(* Logix 5000 project; controller Generic 1768-L43 rev 15.6; software revision 15.01; part 4 of 10 *)
(* tags used below, declared in another part *)
   EL_CTRL_7 : UDT_AxisHistory_CTRL;
   EL_CTRL_8 : UDT_AxisHistory_CTRL;
   EventLog_N7 : UDT_AxisHistory_DLM[51];
   EventLog_N8 : UDT_AxisHistory_DLM[51];
   LogLength : DINT;
   Motion_Group : ALIAS FOR MotionGroup;
   Servo_Axis_Node_7 : ALIAS FOR AXIS_Servo_Generic;
   Servo_Axis_Node_8 : ALIAS FOR AXIS_Servo_Generic;
(* AXIS_EventLog, continued *)

ROUTINE R07_EventLog_Node7   (* ladder *)
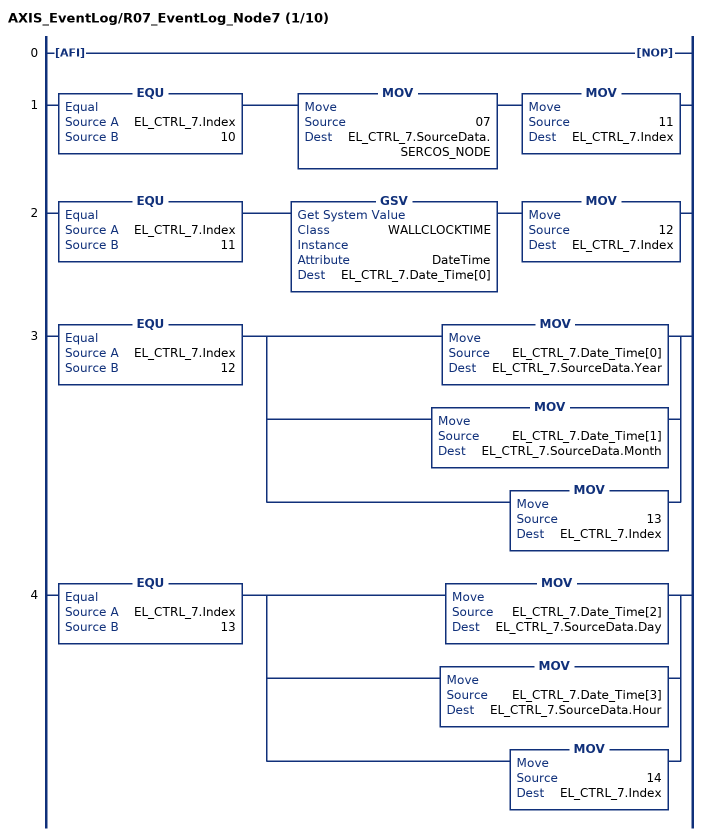
   0: AFI()NOP();
   1: EQU(EL_CTRL_7.Index,10)MOV(07,EL_CTRL_7.SourceData.SERCOS_NODE)MOV(11,EL_CTRL_7.Index);
   2: EQU(EL_CTRL_7.Index,11)GSV(WALLCLOCKTIME,,DateTime,EL_CTRL_7.Date_Time[0])MOV(12,EL_CTRL_7.Index);
   3: EQU(EL_CTRL_7.Index,12)[MOV(EL_CTRL_7.Date_Time[0],EL_CTRL_7.SourceData.Year) ,MOV(EL_CTRL_7.Date_Time[1],EL_CTRL_7.SourceData.Month) ,MOV(13,EL_CTRL_7.Index) ];
   4: EQU(EL_CTRL_7.Index,13)[MOV(EL_CTRL_7.Date_Time[2],EL_CTRL_7.SourceData.Day) ,MOV(EL_CTRL_7.Date_Time[3],EL_CTRL_7.SourceData.Hour) ,MOV(14,EL_CTRL_7.Index) ];
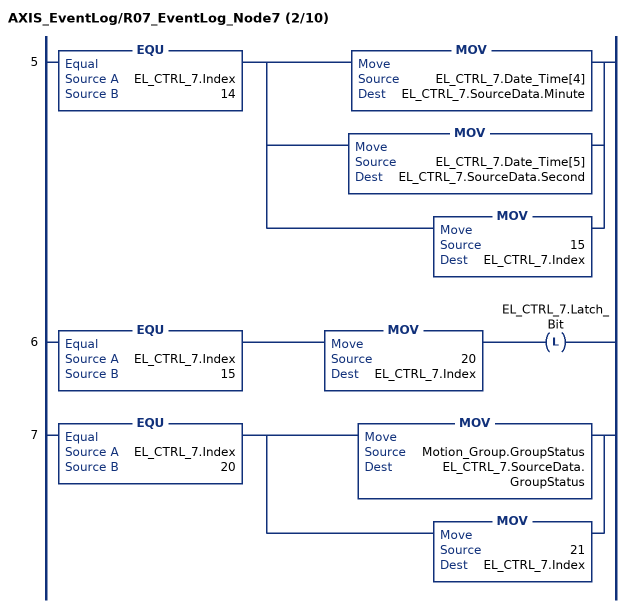
   5: EQU(EL_CTRL_7.Index,14)[MOV(EL_CTRL_7.Date_Time[4],EL_CTRL_7.SourceData.Minute) ,MOV(EL_CTRL_7.Date_Time[5],EL_CTRL_7.SourceData.Second) ,MOV(15,EL_CTRL_7.Index) ];
   6: EQU(EL_CTRL_7.Index,15)MOV(20,EL_CTRL_7.Index)OTL(EL_CTRL_7.Latch_Bit);
   7: EQU(EL_CTRL_7.Index,20)[MOV(Motion_Group.GroupStatus,EL_CTRL_7.SourceData.GroupStatus) ,MOV(21,EL_CTRL_7.Index) ];
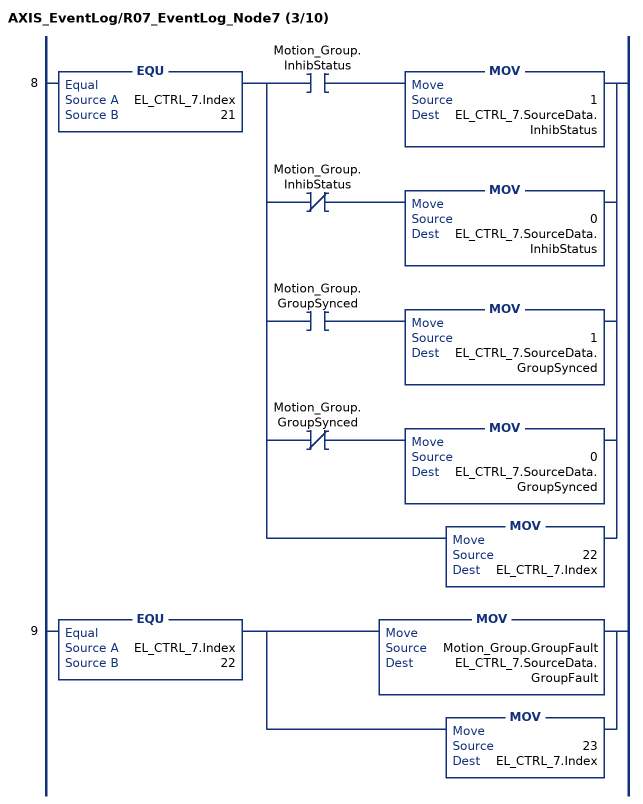
   8: EQU(EL_CTRL_7.Index,21)[XIC(Motion_Group.InhibStatus) MOV(1,EL_CTRL_7.SourceData.InhibStatus) ,XIO(Motion_Group.InhibStatus) MOV(0,EL_CTRL_7.SourceData.InhibStatus) ,XIC(Motion_Group.GroupSynced) MOV(1,EL_CTRL_7.SourceData.GroupSynced) ,XIO(Motion_Group.GroupSynced) MOV(0,EL_CTRL_7.SourceData.GroupSynced) ,MOV(22,EL_CTRL_7.Index) ];
   9: EQU(EL_CTRL_7.Index,22)[MOV(Motion_Group.GroupFault,EL_CTRL_7.SourceData.GroupFault) ,MOV(23,EL_CTRL_7.Index) ];
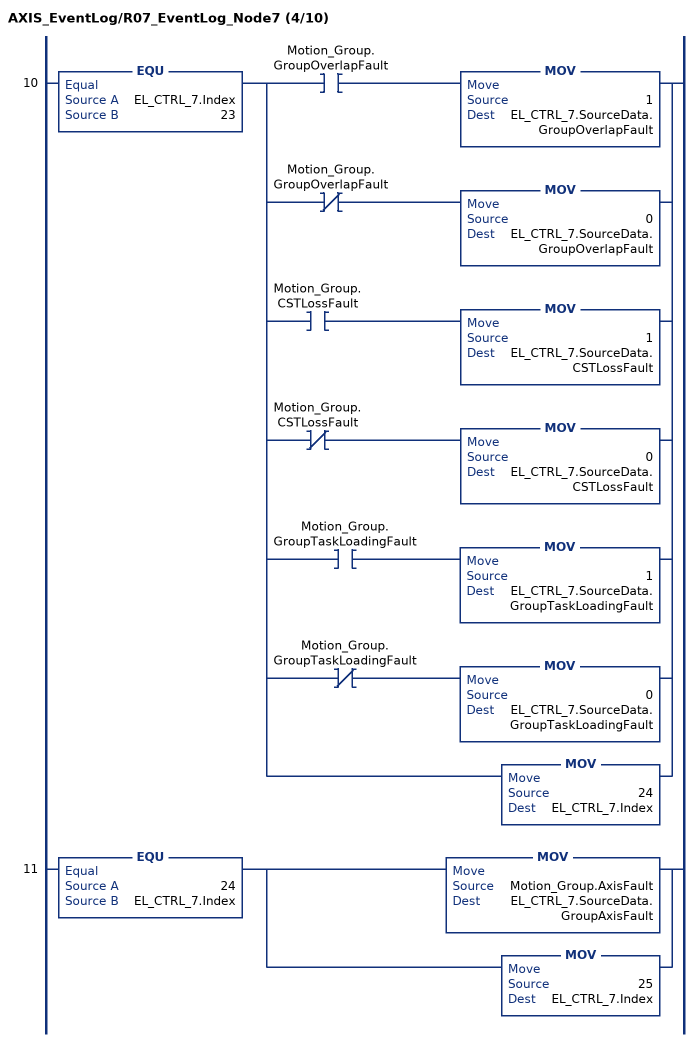
   10: EQU(EL_CTRL_7.Index,23)[XIC(Motion_Group.GroupOverlapFault) MOV(1,EL_CTRL_7.SourceData.GroupOverlapFault) ,XIO(Motion_Group.GroupOverlapFault) MOV(0,EL_CTRL_7.SourceData.GroupOverlapFault) ,XIC(Motion_Group.CSTLossFault) MOV(1,EL_CTRL_7.SourceData.CSTLossFault) ,XIO(Motion_Group.CSTLossFault) MOV(0,EL_CTRL_7.SourceData.CSTLossFault) ,XIC(Motion_Group.GroupTaskLoadingFault) MOV(1,EL_CTRL_7.SourceData.GroupTaskLoadingFault) ,XIO(Motion_Group.GroupTaskLoadingFault) MOV(0,EL_CTRL_7.SourceData.GroupTaskLoadingFault) ,MOV(24,EL_CTRL_7.Index) ];
   11: EQU(24,EL_CTRL_7.Index)[MOV(Motion_Group.AxisFault,EL_CTRL_7.SourceData.GroupAxisFault) ,MOV(25,EL_CTRL_7.Index) ];
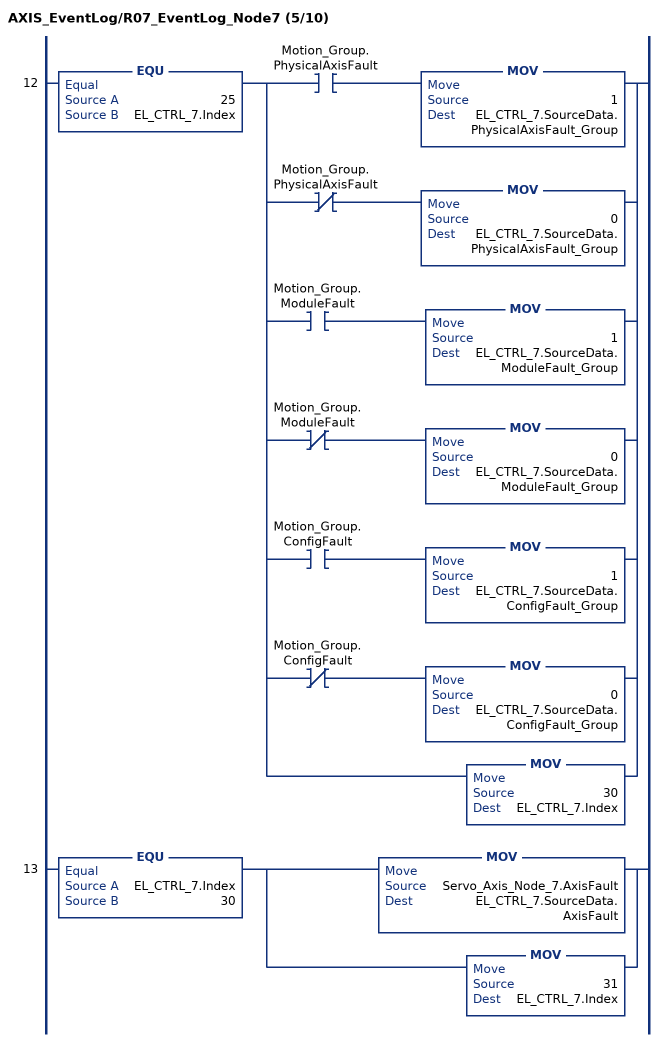
   12: EQU(25,EL_CTRL_7.Index)[XIC(Motion_Group.PhysicalAxisFault) MOV(1,EL_CTRL_7.SourceData.PhysicalAxisFault_Group) ,XIO(Motion_Group.PhysicalAxisFault) MOV(0,EL_CTRL_7.SourceData.PhysicalAxisFault_Group) ,XIC(Motion_Group.ModuleFault) MOV(1,EL_CTRL_7.SourceData.ModuleFault_Group) ,XIO(Motion_Group.ModuleFault) MOV(0,EL_CTRL_7.SourceData.ModuleFault_Group) ,XIC(Motion_Group.ConfigFault) MOV(1,EL_CTRL_7.SourceData.ConfigFault_Group) ,XIO(Motion_Group.ConfigFault) MOV(0,EL_CTRL_7.SourceData.ConfigFault_Group) ,MOV(30,EL_CTRL_7.Index) ];
   13: EQU(EL_CTRL_7.Index,30)[MOV(Servo_Axis_Node_7.AxisFault,EL_CTRL_7.SourceData.AxisFault) ,MOV(31,EL_CTRL_7.Index) ];
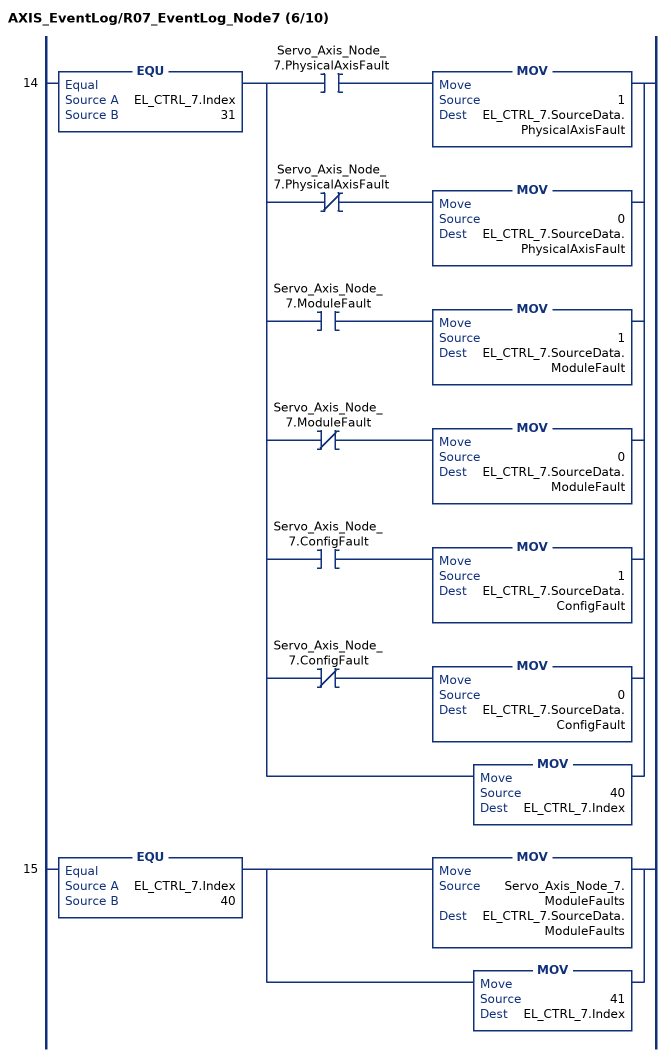
   14: EQU(EL_CTRL_7.Index,31)[XIC(Servo_Axis_Node_7.PhysicalAxisFault) MOV(1,EL_CTRL_7.SourceData.PhysicalAxisFault) ,XIO(Servo_Axis_Node_7.PhysicalAxisFault) MOV(0,EL_CTRL_7.SourceData.PhysicalAxisFault) ,XIC(Servo_Axis_Node_7.ModuleFault) MOV(1,EL_CTRL_7.SourceData.ModuleFault) ,XIO(Servo_Axis_Node_7.ModuleFault) MOV(0,EL_CTRL_7.SourceData.ModuleFault) ,XIC(Servo_Axis_Node_7.ConfigFault) MOV(1,EL_CTRL_7.SourceData.ConfigFault) ,XIO(Servo_Axis_Node_7.ConfigFault) MOV(0,EL_CTRL_7.SourceData.ConfigFault) ,MOV(40,EL_CTRL_7.Index) ];
   15: EQU(EL_CTRL_7.Index,40)[MOV(Servo_Axis_Node_7.ModuleFaults,EL_CTRL_7.SourceData.ModuleFaults) ,MOV(41,EL_CTRL_7.Index) ];
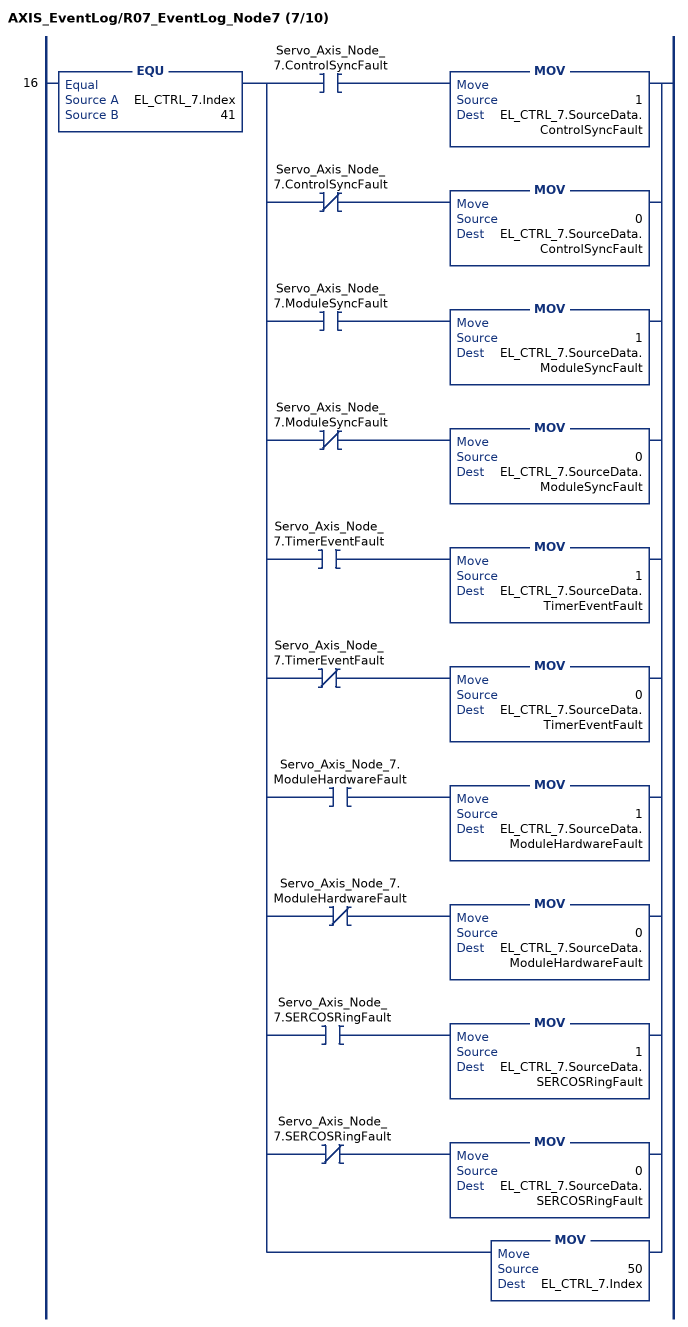
   16: EQU(EL_CTRL_7.Index,41)[XIC(Servo_Axis_Node_7.ControlSyncFault) MOV(1,EL_CTRL_7.SourceData.ControlSyncFault) ,XIO(Servo_Axis_Node_7.ControlSyncFault) MOV(0,EL_CTRL_7.SourceData.ControlSyncFault) ,XIC(Servo_Axis_Node_7.ModuleSyncFault) MOV(1,EL_CTRL_7.SourceData.ModuleSyncFault) ,XIO(Servo_Axis_Node_7.ModuleSyncFault) MOV(0,EL_CTRL_7.SourceData.ModuleSyncFault) ,XIC(Servo_Axis_Node_7.TimerEventFault) MOV(1,EL_CTRL_7.SourceData.TimerEventFault) ,XIO(Servo_Axis_Node_7.TimerEventFault) MOV(0,EL_CTRL_7.SourceData.TimerEventFault) ,XIC(Servo_Axis_Node_7.ModuleHardwareFault) MOV(1,EL_CTRL_7.SourceData.ModuleHardwareFault) ,XIO(Servo_Axis_Node_7.ModuleHardwareFault) MOV(0,EL_CTRL_7.SourceData.ModuleHardwareFault) ,XIC(Servo_Axis_Node_7.SERCOSRingFault) MOV(1,EL_CTRL_7.SourceData.SERCOSRingFault) ,XIO(Servo_Axis_Node_7.SERCOSRingFault) MOV(0,EL_CTRL_7.SourceData.SERCOSRingFault) ,MOV(50,EL_CTRL_7.Index) ];
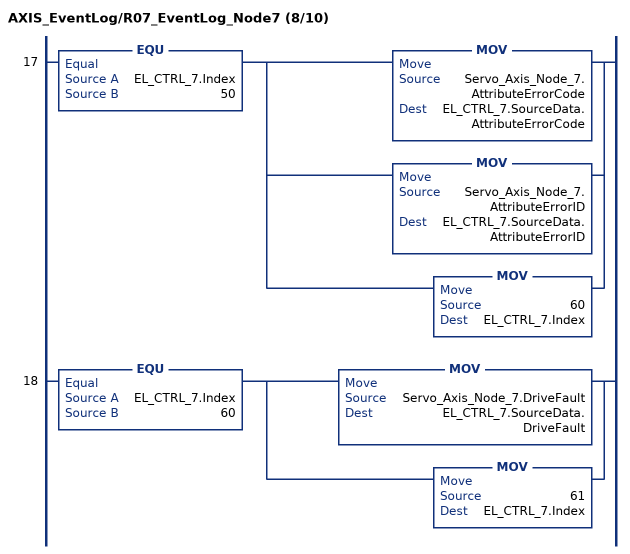
   17: EQU(EL_CTRL_7.Index,50)[MOV(Servo_Axis_Node_7.AttributeErrorCode,EL_CTRL_7.SourceData.AttributeErrorCode) ,MOV(Servo_Axis_Node_7.AttributeErrorID,EL_CTRL_7.SourceData.AttributeErrorID) ,MOV(60,EL_CTRL_7.Index) ];
   18: EQU(EL_CTRL_7.Index,60)[MOV(Servo_Axis_Node_7.DriveFault,EL_CTRL_7.SourceData.DriveFault) ,MOV(61,EL_CTRL_7.Index) ];
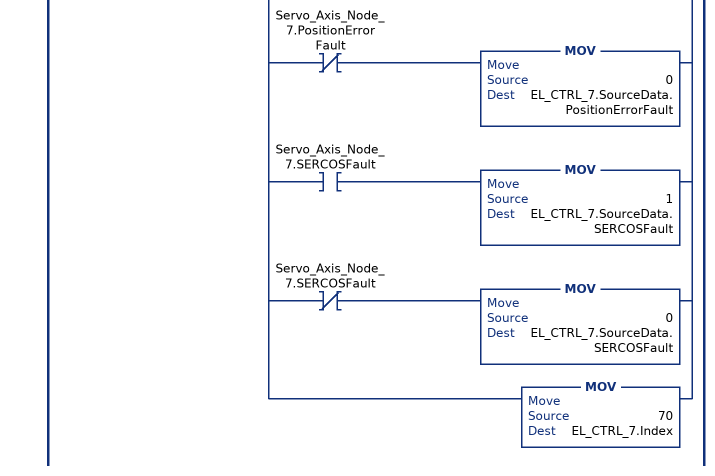
   19: EQU(EL_CTRL_7.Index,61)[XIC(Servo_Axis_Node_7.PosSoftOvertravelFault) MOV(1,EL_CTRL_7.SourceData.PosSoftOvertravelFault) ,XIO(Servo_Axis_Node_7.PosSoftOvertravelFault) MOV(0,EL_CTRL_7.SourceData.PosSoftOvertravelFault) ,XIC(Servo_Axis_Node_7.NegSoftOvertravelFault) MOV(1,EL_CTRL_7.SourceData.NegSoftOvertravelFault) ,XIO(Servo_Axis_Node_7.NegSoftOvertravelFault) MOV(0,EL_CTRL_7.SourceData.NegSoftOvertravelFault) ,XIC(Servo_Axis_Node_7.PosHardOvertravelFault) MOV(1,EL_CTRL_7.SourceData.PosHardOvertravelFault) ,XIO(Servo_Axis_Node_7.PosHardOvertravelFault) MOV(0,EL_CTRL_7.SourceData.PosHardOvertravelFault) ,XIC(Servo_Axis_Node_7.NegHardOvertravelFault) MOV(1,EL_CTRL_7.SourceData.NegHardOvertravelFault) ,XIO(Servo_Axis_Node_7.NegHardOvertravelFault) MOV(0,EL_CTRL_7.SourceData.NegHardOvertravelFault) ,XIC(Servo_Axis_Node_7.MotFeedbackFault) MOV(1,EL_CTRL_7.SourceData.MotFeedbackFault) ,XIO(Servo_Axis_Node_7.MotFeedbackFault) MOV(0,EL_CTRL_7.SourceData.MotFeedbackFault) ,XIC(Servo_Axis_Node_7.MotFeedbackNoiseFault) MOV(1,EL_CTRL_7.SourceData.MotFeedbackNoiseFault) ,XIO(Servo_Axis_Node_7.MotFeedbackNoiseFault) MOV(0,EL_CTRL_7.SourceData.MotFeedbackNoiseFault) ,XIC(Servo_Axis_Node_7.AuxFeedbackFault) MOV(1,EL_CTRL_7.SourceData.AuxFeedbackFault) ,XIO(Servo_Axis_Node_7.AuxFeedbackFault) MOV(0,EL_CTRL_7.SourceData.AuxFeedbackFault) ,XIC(Servo_Axis_Node_7.AuxFeedbackNoiseFault) MOV(1,EL_CTRL_7.SourceData.AuxFeedbackNoiseFault) ,XIO(Servo_Axis_Node_7.AuxFeedbackNoiseFault) MOV(0,EL_CTRL_7.SourceData.AuxFeedbackNoiseFault) ,XIC(Servo_Axis_Node_7.DriveEnableInputFault) MOV(1,EL_CTRL_7.SourceData.DriveEnableInputFault) ,XIO(Servo_Axis_Node_7.DriveEnableInputFault) MOV(0,EL_CTRL_7.SourceData.DriveEnableInputFault) ,XIC(Servo_Axis_Node_7.CommonBusFault) MOV(1,EL_CTRL_7.SourceData.CommonBusFault) ,XIO(Servo_Axis_Node_7.CommonBusFault) MOV(0,EL_CTRL_7.SourceData.CommonBusFault) ,XIC(Servo_Axis_Node_7.PreChargeOverloadFault) MOV(1,EL_CTRL_7.SourceData.PreChargeOverloadFault) ,XIO(Servo_Axis_Node_7.PreChargeOverloadFault) MOV(0,EL_CTRL_7.SourceData.PreChargeOverloadFault) ,XIC(Servo_Axis_Node_7.GroundShortFault) MOV(1,EL_CTRL_7.SourceData.GroundShortFault) ,XIO(Servo_Axis_Node_7.GroundShortFault) MOV(0,EL_CTRL_7.SourceData.GroundShortFault) ,XIC(Servo_Axis_Node_7.DriveHardFault) MOV(1,EL_CTRL_7.SourceData.DriveHardFault) ,XIO(Servo_Axis_Node_7.DriveHardFault) MOV(0,EL_CTRL_7.SourceData.DriveHardFault) ,XIC(Servo_Axis_Node_7.OverSpeedFault) MOV(1,EL_CTRL_7.SourceData.OverSpeedFault) ,XIO(Servo_Axis_Node_7.OverSpeedFault) MOV(0,EL_CTRL_7.SourceData.OverSpeedFault) ,XIC(Servo_Axis_Node_7.OverloadFault) MOV(1,EL_CTRL_7.SourceData.OverloadFault) ,XIO(Servo_Axis_Node_7.OverloadFault) MOV(0,EL_CTRL_7.SourceData.OverloadFault) ,XIC(Servo_Axis_Node_7.DriveOvertempFault) MOV(1,EL_CTRL_7.SourceData.DriveOvertempFault) ,XIO(Servo_Axis_Node_7.DriveOvertempFault) MOV(0,EL_CTRL_7.SourceData.DriveOvertempFault) ,XIC(Servo_Axis_Node_7.MotorOvertempFault) MOV(1,EL_CTRL_7.SourceData.MotorOvertempFault) ,XIO(Servo_Axis_Node_7.MotorOvertempFault) MOV(0,EL_CTRL_7.SourceData.MotorOvertempFault) ,XIC(Servo_Axis_Node_7.DriveCoolingFault) MOV(1,EL_CTRL_7.SourceData.DriveCoolingFault) ,XIO(Servo_Axis_Node_7.DriveCoolingFault) MOV(0,EL_CTRL_7.SourceData.DriveCoolingFault) ,XIC(Servo_Axis_Node_7.DriveControlVoltageFault) MOV(1,EL_CTRL_7.SourceData.DriveControlVoltageFault) ,XIO(Servo_Axis_Node_7.DriveControlVoltageFault) MOV(0,EL_CTRL_7.SourceData.DriveControlVoltageFault) ,XIC(Servo_Axis_Node_7.FeedbackFault) MOV(1,EL_CTRL_7.SourceData.FeedbackFault) ,XIO(Servo_Axis_Node_7.FeedbackFault) MOV(0,EL_CTRL_7.SourceData.FeedbackFault) ,XIC(Servo_Axis_Node_7.CommutationFault) MOV(1,EL_CTRL_7.SourceData.CommutationFault) ,XIO(Servo_Axis_Node_7.CommutationFault) MOV(0,EL_CTRL_7.SourceData.CommutationFault) ,XIC(Servo_Axis_Node_7.DriveOvercurrentFault) MOV(1,EL_CTRL_7.SourceData.DriveOvercurrentFault) ,XIO(Servo_Axis_Node_7.DriveOvercurrentFault) MOV(0,EL_CTRL_7.SourceData.DriveOvercurrentFault) ,XIC(Servo_Axis_Node_7.DriveOvervoltageFault) MOV(1,EL_CTRL_7.SourceData.DriveOvervoltageFault) ,XIO(Servo_Axis_Node_7.DriveOvervoltageFault) MOV(0,EL_CTRL_7.SourceData.DriveOvervoltageFault) ,XIC(Servo_Axis_Node_7.DriveUndervoltageFault) MOV(1,EL_CTRL_7.SourceData.DriveUndervoltageFault) ,XIO(Servo_Axis_Node_7.DriveUndervoltageFault) MOV(0,EL_CTRL_7.SourceData.DriveUndervoltageFault) ,XIC(Servo_Axis_Node_7.PowerPhaseLossFault) MOV(1,EL_CTRL_7.SourceData.PowerPhaseLossFault) ,XIO(Servo_Axis_Node_7.PowerPhaseLossFault) MOV(0,EL_CTRL_7.SourceData.PowerPhaseLossFault) ,XIC(Servo_Axis_Node_7.PositionErrorFault) MOV(1,EL_CTRL_7.SourceData.PositionErrorFault) ,XIO(Servo_Axis_Node_7.PositionErrorFault) MOV(0,EL_CTRL_7.SourceData.PositionErrorFault) ,XIC(Servo_Axis_Node_7.SERCOSFault) MOV(1,EL_CTRL_7.SourceData.SERCOSFault) ,XIO(Servo_Axis_Node_7.SERCOSFault) MOV(0,EL_CTRL_7.SourceData.SERCOSFault) ,MOV(70,EL_CTRL_7.Index) ];
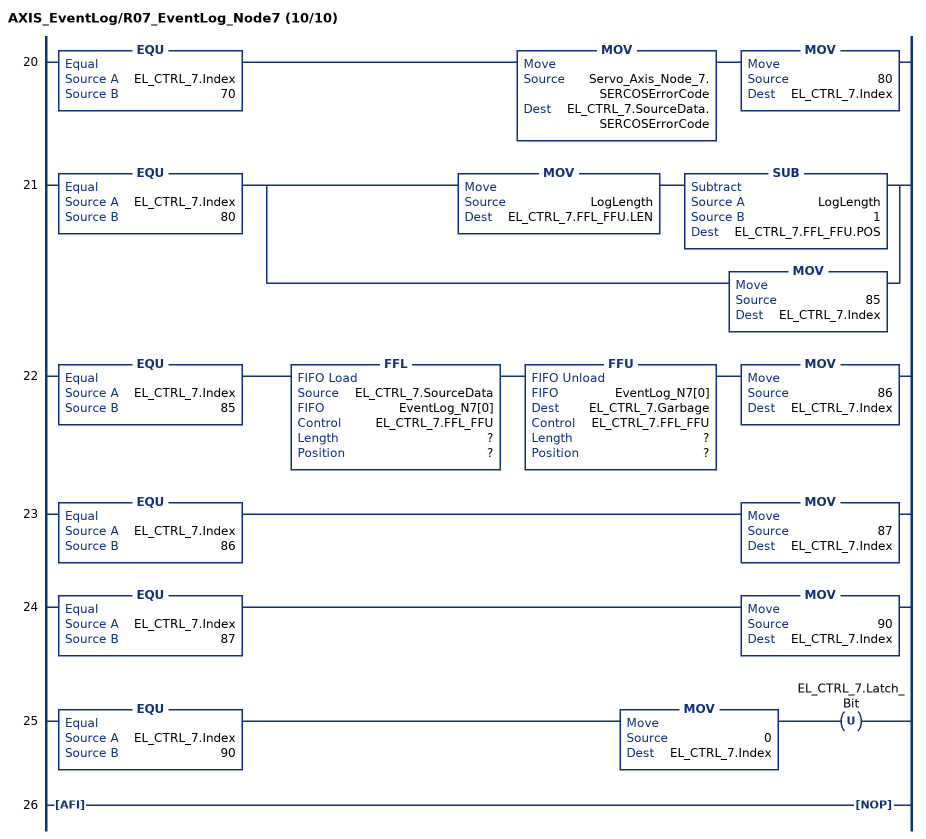
   20: EQU(EL_CTRL_7.Index,70)MOV(Servo_Axis_Node_7.SERCOSErrorCode,EL_CTRL_7.SourceData.SERCOSErrorCode)MOV(80,EL_CTRL_7.Index);
   21: EQU(EL_CTRL_7.Index,80)[MOV(LogLength,EL_CTRL_7.FFL_FFU.LEN) SUB(LogLength,1,EL_CTRL_7.FFL_FFU.POS) ,MOV(85,EL_CTRL_7.Index) ];
   22: EQU(EL_CTRL_7.Index,85)FFL(EL_CTRL_7.SourceData,EventLog_N7[0],EL_CTRL_7.FFL_FFU,?,?)FFU(EventLog_N7[0],EL_CTRL_7.Garbage,EL_CTRL_7.FFL_FFU,?,?)MOV(86,EL_CTRL_7.Index);
   23: EQU(EL_CTRL_7.Index,86)MOV(87,EL_CTRL_7.Index);
   24: EQU(EL_CTRL_7.Index,87)MOV(90,EL_CTRL_7.Index);
   25: EQU(EL_CTRL_7.Index,90)MOV(0,EL_CTRL_7.Index)OTU(EL_CTRL_7.Latch_Bit);
   26: AFI()NOP();
END_ROUTINE

ROUTINE R08_EventLog_Node8   (* ladder *)
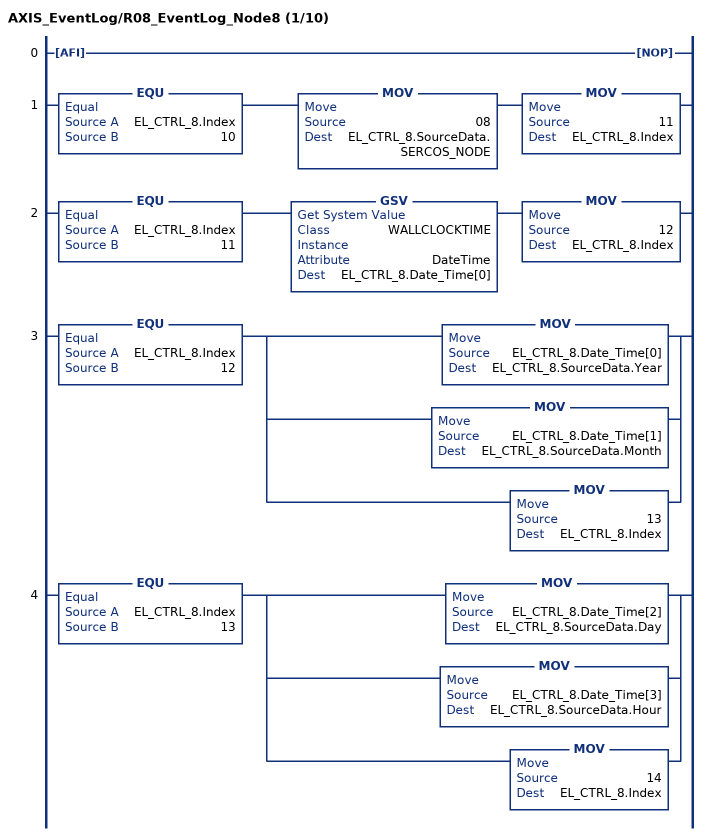
   0: AFI()NOP();
   1: EQU(EL_CTRL_8.Index,10)MOV(08,EL_CTRL_8.SourceData.SERCOS_NODE)MOV(11,EL_CTRL_8.Index);
   2: EQU(EL_CTRL_8.Index,11)GSV(WALLCLOCKTIME,,DateTime,EL_CTRL_8.Date_Time[0])MOV(12,EL_CTRL_8.Index);
   3: EQU(EL_CTRL_8.Index,12)[MOV(EL_CTRL_8.Date_Time[0],EL_CTRL_8.SourceData.Year) ,MOV(EL_CTRL_8.Date_Time[1],EL_CTRL_8.SourceData.Month) ,MOV(13,EL_CTRL_8.Index) ];
   4: EQU(EL_CTRL_8.Index,13)[MOV(EL_CTRL_8.Date_Time[2],EL_CTRL_8.SourceData.Day) ,MOV(EL_CTRL_8.Date_Time[3],EL_CTRL_8.SourceData.Hour) ,MOV(14,EL_CTRL_8.Index) ];
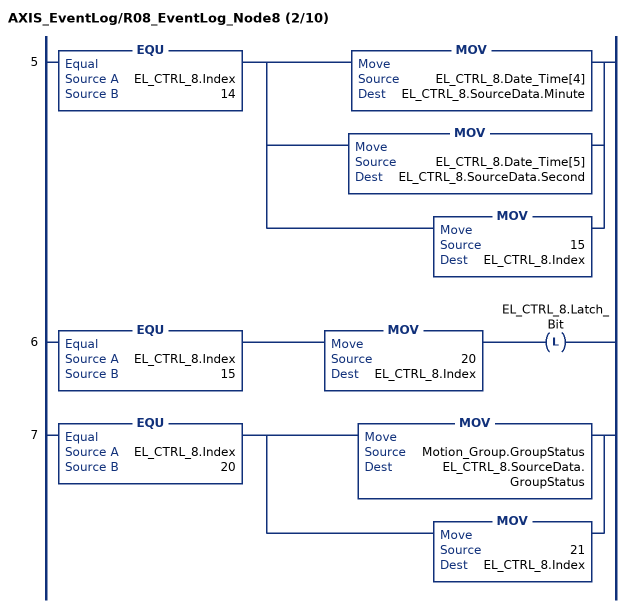
   5: EQU(EL_CTRL_8.Index,14)[MOV(EL_CTRL_8.Date_Time[4],EL_CTRL_8.SourceData.Minute) ,MOV(EL_CTRL_8.Date_Time[5],EL_CTRL_8.SourceData.Second) ,MOV(15,EL_CTRL_8.Index) ];
   6: EQU(EL_CTRL_8.Index,15)MOV(20,EL_CTRL_8.Index)OTL(EL_CTRL_8.Latch_Bit);
   7: EQU(EL_CTRL_8.Index,20)[MOV(Motion_Group.GroupStatus,EL_CTRL_8.SourceData.GroupStatus) ,MOV(21,EL_CTRL_8.Index) ];
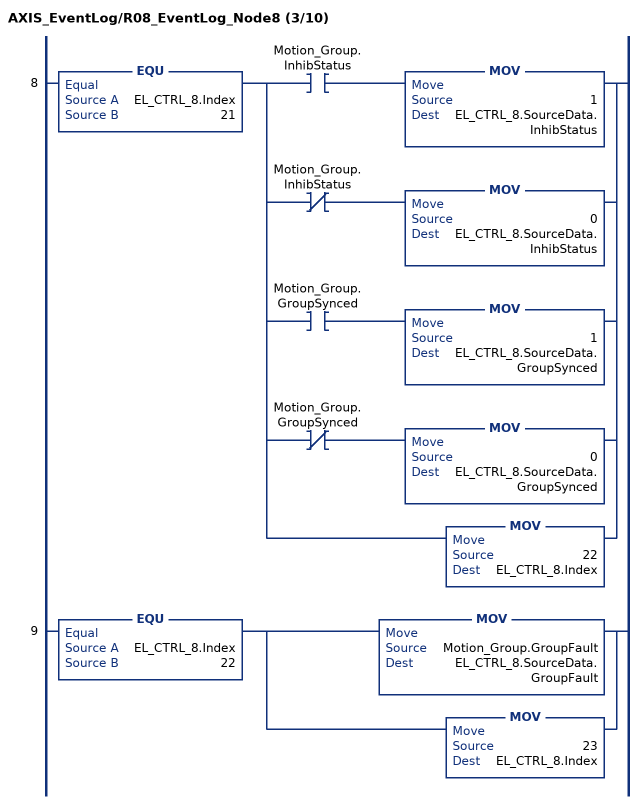
   8: EQU(EL_CTRL_8.Index,21)[XIC(Motion_Group.InhibStatus) MOV(1,EL_CTRL_8.SourceData.InhibStatus) ,XIO(Motion_Group.InhibStatus) MOV(0,EL_CTRL_8.SourceData.InhibStatus) ,XIC(Motion_Group.GroupSynced) MOV(1,EL_CTRL_8.SourceData.GroupSynced) ,XIO(Motion_Group.GroupSynced) MOV(0,EL_CTRL_8.SourceData.GroupSynced) ,MOV(22,EL_CTRL_8.Index) ];
   9: EQU(EL_CTRL_8.Index,22)[MOV(Motion_Group.GroupFault,EL_CTRL_8.SourceData.GroupFault) ,MOV(23,EL_CTRL_8.Index) ];
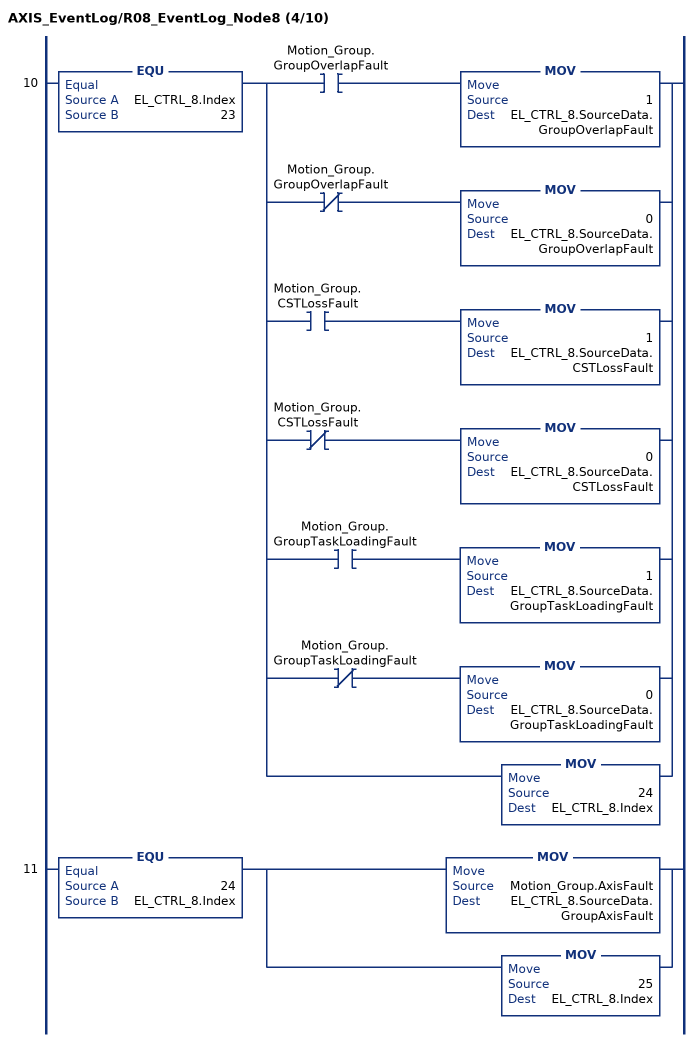
   10: EQU(EL_CTRL_8.Index,23)[XIC(Motion_Group.GroupOverlapFault) MOV(1,EL_CTRL_8.SourceData.GroupOverlapFault) ,XIO(Motion_Group.GroupOverlapFault) MOV(0,EL_CTRL_8.SourceData.GroupOverlapFault) ,XIC(Motion_Group.CSTLossFault) MOV(1,EL_CTRL_8.SourceData.CSTLossFault) ,XIO(Motion_Group.CSTLossFault) MOV(0,EL_CTRL_8.SourceData.CSTLossFault) ,XIC(Motion_Group.GroupTaskLoadingFault) MOV(1,EL_CTRL_8.SourceData.GroupTaskLoadingFault) ,XIO(Motion_Group.GroupTaskLoadingFault) MOV(0,EL_CTRL_8.SourceData.GroupTaskLoadingFault) ,MOV(24,EL_CTRL_8.Index) ];
   11: EQU(24,EL_CTRL_8.Index)[MOV(Motion_Group.AxisFault,EL_CTRL_8.SourceData.GroupAxisFault) ,MOV(25,EL_CTRL_8.Index) ];
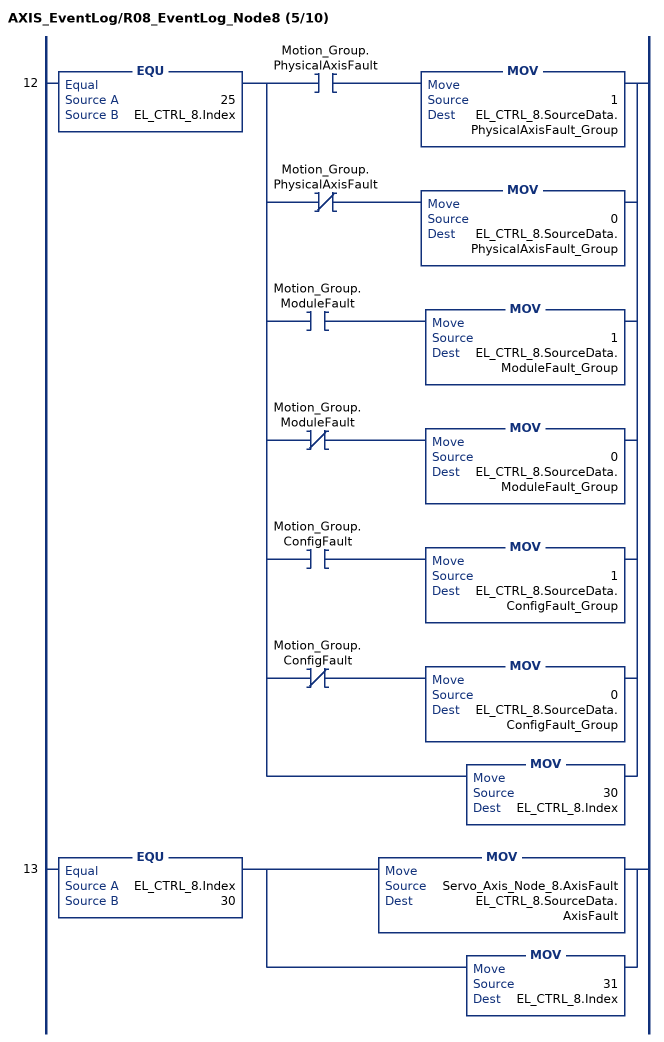
   12: EQU(25,EL_CTRL_8.Index)[XIC(Motion_Group.PhysicalAxisFault) MOV(1,EL_CTRL_8.SourceData.PhysicalAxisFault_Group) ,XIO(Motion_Group.PhysicalAxisFault) MOV(0,EL_CTRL_8.SourceData.PhysicalAxisFault_Group) ,XIC(Motion_Group.ModuleFault) MOV(1,EL_CTRL_8.SourceData.ModuleFault_Group) ,XIO(Motion_Group.ModuleFault) MOV(0,EL_CTRL_8.SourceData.ModuleFault_Group) ,XIC(Motion_Group.ConfigFault) MOV(1,EL_CTRL_8.SourceData.ConfigFault_Group) ,XIO(Motion_Group.ConfigFault) MOV(0,EL_CTRL_8.SourceData.ConfigFault_Group) ,MOV(30,EL_CTRL_8.Index) ];
   13: EQU(EL_CTRL_8.Index,30)[MOV(Servo_Axis_Node_8.AxisFault,EL_CTRL_8.SourceData.AxisFault) ,MOV(31,EL_CTRL_8.Index) ];
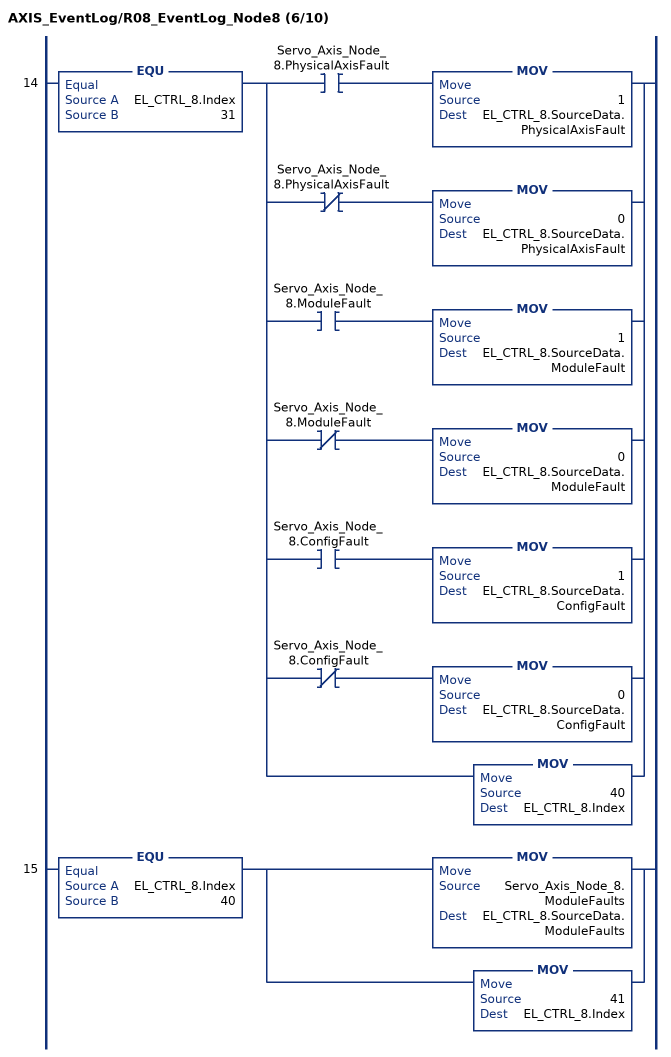
   14: EQU(EL_CTRL_8.Index,31)[XIC(Servo_Axis_Node_8.PhysicalAxisFault) MOV(1,EL_CTRL_8.SourceData.PhysicalAxisFault) ,XIO(Servo_Axis_Node_8.PhysicalAxisFault) MOV(0,EL_CTRL_8.SourceData.PhysicalAxisFault) ,XIC(Servo_Axis_Node_8.ModuleFault) MOV(1,EL_CTRL_8.SourceData.ModuleFault) ,XIO(Servo_Axis_Node_8.ModuleFault) MOV(0,EL_CTRL_8.SourceData.ModuleFault) ,XIC(Servo_Axis_Node_8.ConfigFault) MOV(1,EL_CTRL_8.SourceData.ConfigFault) ,XIO(Servo_Axis_Node_8.ConfigFault) MOV(0,EL_CTRL_8.SourceData.ConfigFault) ,MOV(40,EL_CTRL_8.Index) ];
   15: EQU(EL_CTRL_8.Index,40)[MOV(Servo_Axis_Node_8.ModuleFaults,EL_CTRL_8.SourceData.ModuleFaults) ,MOV(41,EL_CTRL_8.Index) ];
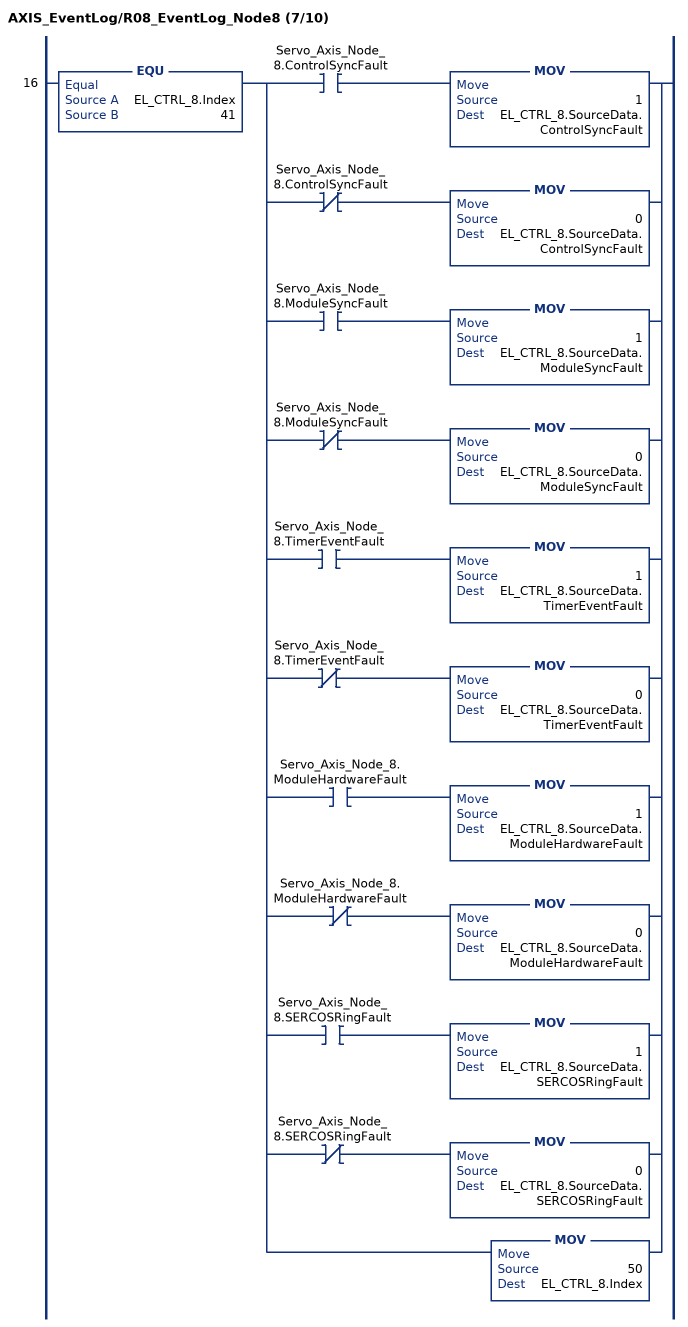
   16: EQU(EL_CTRL_8.Index,41)[XIC(Servo_Axis_Node_8.ControlSyncFault) MOV(1,EL_CTRL_8.SourceData.ControlSyncFault) ,XIO(Servo_Axis_Node_8.ControlSyncFault) MOV(0,EL_CTRL_8.SourceData.ControlSyncFault) ,XIC(Servo_Axis_Node_8.ModuleSyncFault) MOV(1,EL_CTRL_8.SourceData.ModuleSyncFault) ,XIO(Servo_Axis_Node_8.ModuleSyncFault) MOV(0,EL_CTRL_8.SourceData.ModuleSyncFault) ,XIC(Servo_Axis_Node_8.TimerEventFault) MOV(1,EL_CTRL_8.SourceData.TimerEventFault) ,XIO(Servo_Axis_Node_8.TimerEventFault) MOV(0,EL_CTRL_8.SourceData.TimerEventFault) ,XIC(Servo_Axis_Node_8.ModuleHardwareFault) MOV(1,EL_CTRL_8.SourceData.ModuleHardwareFault) ,XIO(Servo_Axis_Node_8.ModuleHardwareFault) MOV(0,EL_CTRL_8.SourceData.ModuleHardwareFault) ,XIC(Servo_Axis_Node_8.SERCOSRingFault) MOV(1,EL_CTRL_8.SourceData.SERCOSRingFault) ,XIO(Servo_Axis_Node_8.SERCOSRingFault) MOV(0,EL_CTRL_8.SourceData.SERCOSRingFault) ,MOV(50,EL_CTRL_8.Index) ];
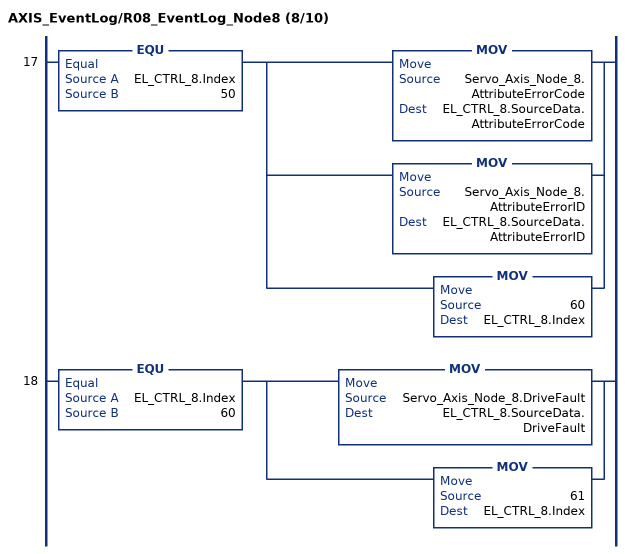
   17: EQU(EL_CTRL_8.Index,50)[MOV(Servo_Axis_Node_8.AttributeErrorCode,EL_CTRL_8.SourceData.AttributeErrorCode) ,MOV(Servo_Axis_Node_8.AttributeErrorID,EL_CTRL_8.SourceData.AttributeErrorID) ,MOV(60,EL_CTRL_8.Index) ];
   18: EQU(EL_CTRL_8.Index,60)[MOV(Servo_Axis_Node_8.DriveFault,EL_CTRL_8.SourceData.DriveFault) ,MOV(61,EL_CTRL_8.Index) ];
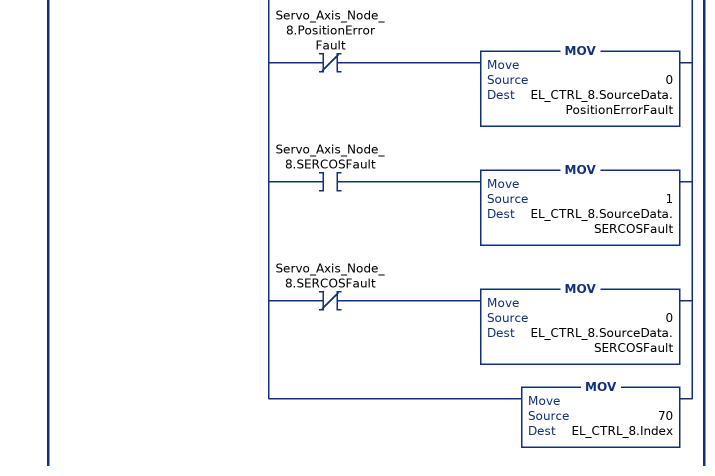
   19: EQU(EL_CTRL_8.Index,61)[XIC(Servo_Axis_Node_8.PosSoftOvertravelFault) MOV(1,EL_CTRL_8.SourceData.PosSoftOvertravelFault) ,XIO(Servo_Axis_Node_8.PosSoftOvertravelFault) MOV(0,EL_CTRL_8.SourceData.PosSoftOvertravelFault) ,XIC(Servo_Axis_Node_8.NegSoftOvertravelFault) MOV(1,EL_CTRL_8.SourceData.NegSoftOvertravelFault) ,XIO(Servo_Axis_Node_8.NegSoftOvertravelFault) MOV(0,EL_CTRL_8.SourceData.NegSoftOvertravelFault) ,XIC(Servo_Axis_Node_8.PosHardOvertravelFault) MOV(1,EL_CTRL_8.SourceData.PosHardOvertravelFault) ,XIO(Servo_Axis_Node_8.PosHardOvertravelFault) MOV(0,EL_CTRL_8.SourceData.PosHardOvertravelFault) ,XIC(Servo_Axis_Node_8.NegHardOvertravelFault) MOV(1,EL_CTRL_8.SourceData.NegHardOvertravelFault) ,XIO(Servo_Axis_Node_8.NegHardOvertravelFault) MOV(0,EL_CTRL_8.SourceData.NegHardOvertravelFault) ,XIC(Servo_Axis_Node_8.MotFeedbackFault) MOV(1,EL_CTRL_8.SourceData.MotFeedbackFault) ,XIO(Servo_Axis_Node_8.MotFeedbackFault) MOV(0,EL_CTRL_8.SourceData.MotFeedbackFault) ,XIC(Servo_Axis_Node_8.MotFeedbackNoiseFault) MOV(1,EL_CTRL_8.SourceData.MotFeedbackNoiseFault) ,XIO(Servo_Axis_Node_8.MotFeedbackNoiseFault) MOV(0,EL_CTRL_8.SourceData.MotFeedbackNoiseFault) ,XIC(Servo_Axis_Node_8.AuxFeedbackFault) MOV(1,EL_CTRL_8.SourceData.AuxFeedbackFault) ,XIO(Servo_Axis_Node_8.AuxFeedbackFault) MOV(0,EL_CTRL_8.SourceData.AuxFeedbackFault) ,XIC(Servo_Axis_Node_8.AuxFeedbackNoiseFault) MOV(1,EL_CTRL_8.SourceData.AuxFeedbackNoiseFault) ,XIO(Servo_Axis_Node_8.AuxFeedbackNoiseFault) MOV(0,EL_CTRL_8.SourceData.AuxFeedbackNoiseFault) ,XIC(Servo_Axis_Node_8.DriveEnableInputFault) MOV(1,EL_CTRL_8.SourceData.DriveEnableInputFault) ,XIO(Servo_Axis_Node_8.DriveEnableInputFault) MOV(0,EL_CTRL_8.SourceData.DriveEnableInputFault) ,XIC(Servo_Axis_Node_8.CommonBusFault) MOV(1,EL_CTRL_8.SourceData.CommonBusFault) ,XIO(Servo_Axis_Node_8.CommonBusFault) MOV(0,EL_CTRL_8.SourceData.CommonBusFault) ,XIC(Servo_Axis_Node_8.PreChargeOverloadFault) MOV(1,EL_CTRL_8.SourceData.PreChargeOverloadFault) ,XIO(Servo_Axis_Node_8.PreChargeOverloadFault) MOV(0,EL_CTRL_8.SourceData.PreChargeOverloadFault) ,XIC(Servo_Axis_Node_8.GroundShortFault) MOV(1,EL_CTRL_8.SourceData.GroundShortFault) ,XIO(Servo_Axis_Node_8.GroundShortFault) MOV(0,EL_CTRL_8.SourceData.GroundShortFault) ,XIC(Servo_Axis_Node_8.DriveHardFault) MOV(1,EL_CTRL_8.SourceData.DriveHardFault) ,XIO(Servo_Axis_Node_8.DriveHardFault) MOV(0,EL_CTRL_8.SourceData.DriveHardFault) ,XIC(Servo_Axis_Node_8.OverSpeedFault) MOV(1,EL_CTRL_8.SourceData.OverSpeedFault) ,XIO(Servo_Axis_Node_8.OverSpeedFault) MOV(0,EL_CTRL_8.SourceData.OverSpeedFault) ,XIC(Servo_Axis_Node_8.OverloadFault) MOV(1,EL_CTRL_8.SourceData.OverloadFault) ,XIO(Servo_Axis_Node_8.OverloadFault) MOV(0,EL_CTRL_8.SourceData.OverloadFault) ,XIC(Servo_Axis_Node_8.DriveOvertempFault) MOV(1,EL_CTRL_8.SourceData.DriveOvertempFault) ,XIO(Servo_Axis_Node_8.DriveOvertempFault) MOV(0,EL_CTRL_8.SourceData.DriveOvertempFault) ,XIC(Servo_Axis_Node_8.MotorOvertempFault) MOV(1,EL_CTRL_8.SourceData.MotorOvertempFault) ,XIO(Servo_Axis_Node_8.MotorOvertempFault) MOV(0,EL_CTRL_8.SourceData.MotorOvertempFault) ,XIC(Servo_Axis_Node_8.DriveCoolingFault) MOV(1,EL_CTRL_8.SourceData.DriveCoolingFault) ,XIO(Servo_Axis_Node_8.DriveCoolingFault) MOV(0,EL_CTRL_8.SourceData.DriveCoolingFault) ,XIC(Servo_Axis_Node_8.DriveControlVoltageFault) MOV(1,EL_CTRL_8.SourceData.DriveControlVoltageFault) ,XIO(Servo_Axis_Node_8.DriveControlVoltageFault) MOV(0,EL_CTRL_8.SourceData.DriveControlVoltageFault) ,XIC(Servo_Axis_Node_8.FeedbackFault) MOV(1,EL_CTRL_8.SourceData.FeedbackFault) ,XIO(Servo_Axis_Node_8.FeedbackFault) MOV(0,EL_CTRL_8.SourceData.FeedbackFault) ,XIC(Servo_Axis_Node_8.CommutationFault) MOV(1,EL_CTRL_8.SourceData.CommutationFault) ,XIO(Servo_Axis_Node_8.CommutationFault) MOV(0,EL_CTRL_8.SourceData.CommutationFault) ,XIC(Servo_Axis_Node_8.DriveOvercurrentFault) MOV(1,EL_CTRL_8.SourceData.DriveOvercurrentFault) ,XIO(Servo_Axis_Node_8.DriveOvercurrentFault) MOV(0,EL_CTRL_8.SourceData.DriveOvercurrentFault) ,XIC(Servo_Axis_Node_8.DriveOvervoltageFault) MOV(1,EL_CTRL_8.SourceData.DriveOvervoltageFault) ,XIO(Servo_Axis_Node_8.DriveOvervoltageFault) MOV(0,EL_CTRL_8.SourceData.DriveOvervoltageFault) ,XIC(Servo_Axis_Node_8.DriveUndervoltageFault) MOV(1,EL_CTRL_8.SourceData.DriveUndervoltageFault) ,XIO(Servo_Axis_Node_8.DriveUndervoltageFault) MOV(0,EL_CTRL_8.SourceData.DriveUndervoltageFault) ,XIC(Servo_Axis_Node_8.PowerPhaseLossFault) MOV(1,EL_CTRL_8.SourceData.PowerPhaseLossFault) ,XIO(Servo_Axis_Node_8.PowerPhaseLossFault) MOV(0,EL_CTRL_8.SourceData.PowerPhaseLossFault) ,XIC(Servo_Axis_Node_8.PositionErrorFault) MOV(1,EL_CTRL_8.SourceData.PositionErrorFault) ,XIO(Servo_Axis_Node_8.PositionErrorFault) MOV(0,EL_CTRL_8.SourceData.PositionErrorFault) ,XIC(Servo_Axis_Node_8.SERCOSFault) MOV(1,EL_CTRL_8.SourceData.SERCOSFault) ,XIO(Servo_Axis_Node_8.SERCOSFault) MOV(0,EL_CTRL_8.SourceData.SERCOSFault) ,MOV(70,EL_CTRL_8.Index) ];
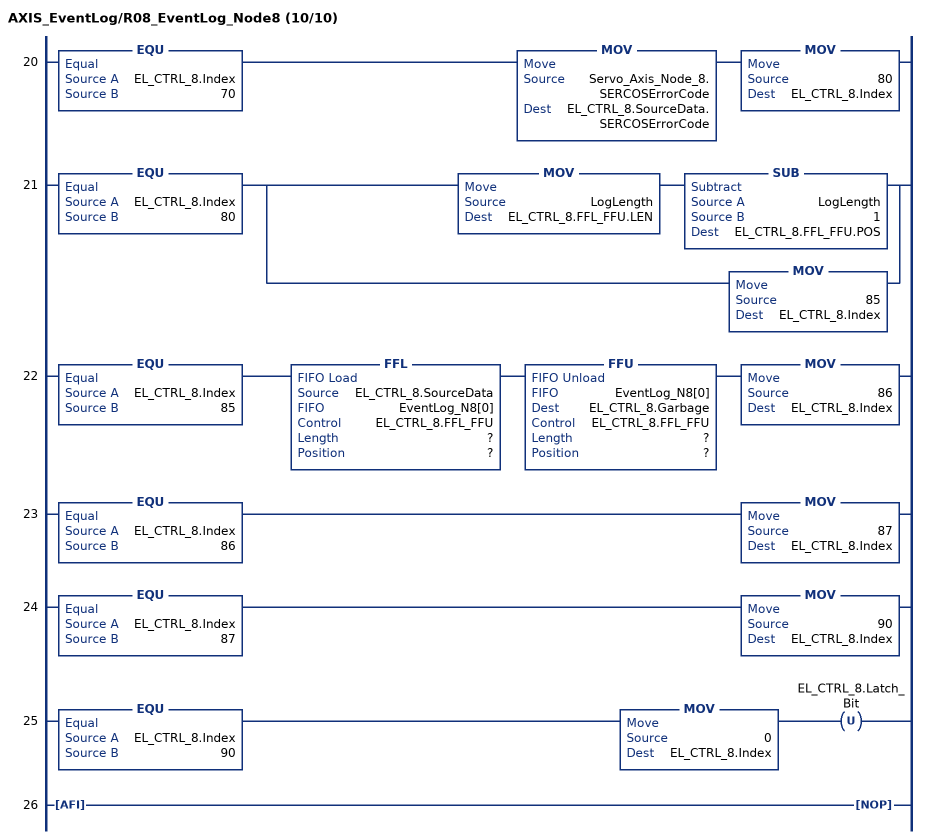
   20: EQU(EL_CTRL_8.Index,70)MOV(Servo_Axis_Node_8.SERCOSErrorCode,EL_CTRL_8.SourceData.SERCOSErrorCode)MOV(80,EL_CTRL_8.Index);
   21: EQU(EL_CTRL_8.Index,80)[MOV(LogLength,EL_CTRL_8.FFL_FFU.LEN) SUB(LogLength,1,EL_CTRL_8.FFL_FFU.POS) ,MOV(85,EL_CTRL_8.Index) ];
   22: EQU(EL_CTRL_8.Index,85)FFL(EL_CTRL_8.SourceData,EventLog_N8[0],EL_CTRL_8.FFL_FFU,?,?)FFU(EventLog_N8[0],EL_CTRL_8.Garbage,EL_CTRL_8.FFL_FFU,?,?)MOV(86,EL_CTRL_8.Index);
   23: EQU(EL_CTRL_8.Index,86)MOV(87,EL_CTRL_8.Index);
   24: EQU(EL_CTRL_8.Index,87)MOV(90,EL_CTRL_8.Index);
   25: EQU(EL_CTRL_8.Index,90)MOV(0,EL_CTRL_8.Index)OTU(EL_CTRL_8.Latch_Bit);
   26: AFI()NOP();
END_ROUTINE
